// Mitsubishi GX Works2 project: Project-2   PLC: Q03UD

PROGRAM MAIN
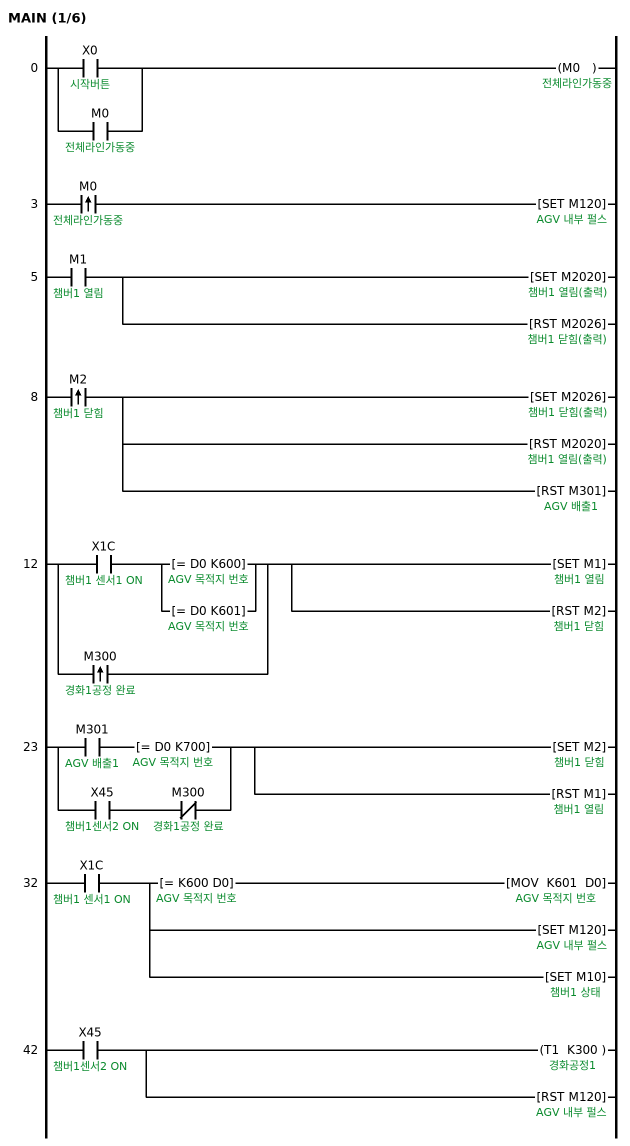
0     LD      X0  ; 시작버튼
      OR      M0  ; 전체라인가동중
      OUT     M0  ; 전체라인가동중
3     LDP     M0  ; 전체라인가동중
      SET     M120  ; AGV 내부 펄스
5     LD      M1  ; 챔버1 열림
      SET     M2020  ; 챔버1 열림(출력)
      RST     M2026  ; 챔버1 닫힘(출력)
8     LDP     M2  ; 챔버1 닫힘
      SET     M2026  ; 챔버1 닫힘(출력)
      RST     M2020  ; 챔버1 열림(출력)
      RST     M301  ; AGV 배출1
12    LD      X1C  ; 챔버1 센서1 ON
      LD=     D0 K600  ; AGV 목적지 번호
      OR=     D0 K601  ; AGV 목적지 번호
      ANB
      ORP     M300  ; 경화1공정 완료
      SET     M1  ; 챔버1 열림
      RST     M2  ; 챔버1 닫힘
23    LD      M301  ; AGV 배출1
      AND=    D0 K700  ; AGV 목적지 번호
      LD      X45  ; 챔버1센서2 ON
      ANI     M300  ; 경화1공정 완료
      ORB
      SET     M2  ; 챔버1 닫힘
      RST     M1  ; 챔버1 열림
32    LD      X1C  ; 챔버1 센서1 ON
      MPS
      AND=    K600 D0  ; AGV 목적지 번호
      MOV     K601 D0
      MPP
      SET     M120  ; AGV 내부 펄스
      SET     M10  ; 챔버1 상태
42    LD      X45  ; 챔버1센서2 ON
      OUT     T1 K300  ; 경화공정1
      RST     M120  ; AGV 내부 펄스
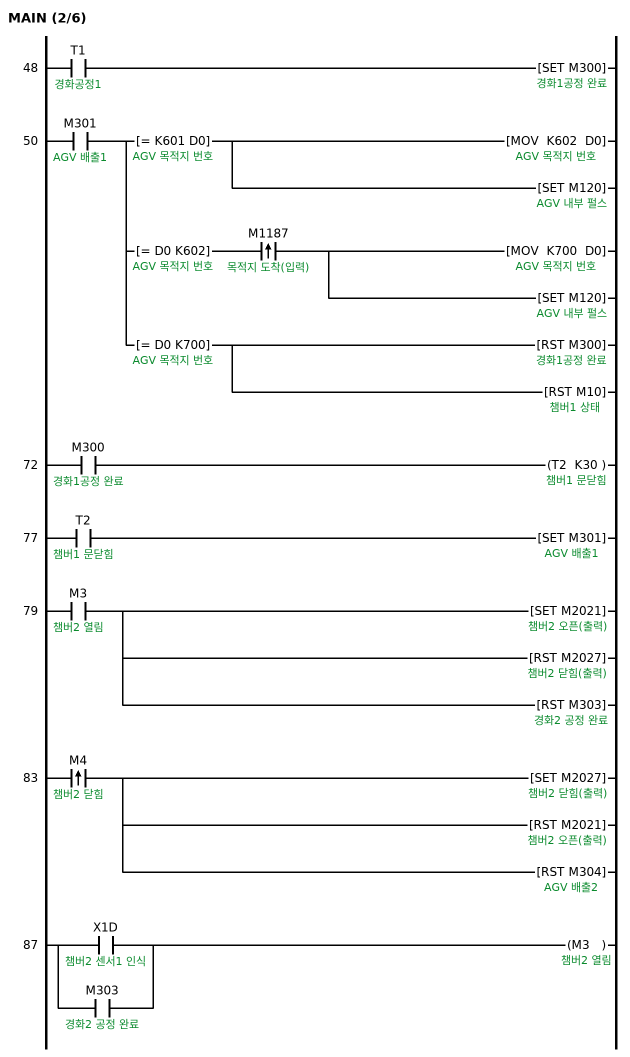
48    LD      T1  ; 경화공정1
      SET     M300  ; 경화1공정 완료
50    LD      M301  ; AGV 배출1
      MPS
      AND=    K601 D0  ; AGV 목적지 번호
      MOV     K602 D0
      SET     M120  ; AGV 내부 펄스
      MRD
      AND=    D0 K602  ; AGV 목적지 번호
      ANDP    M1187  ; 목적지 도착(입력)
      MOV     K700 D0
      SET     M120  ; AGV 내부 펄스
      MPP
      AND=    D0 K700  ; AGV 목적지 번호
      RST     M300  ; 경화1공정 완료
      RST     M10  ; 챔버1 상태
72    LD      M300  ; 경화1공정 완료
      OUT     T2 K30  ; 챔버1 문닫힘
77    LD      T2  ; 챔버1 문닫힘
      SET     M301  ; AGV 배출1
79    LD      M3  ; 챔버2 열림
      SET     M2021  ; 챔버2 오픈(출력)
      RST     M2027  ; 챔버2 닫힘(출력)
      RST     M303  ; 경화2 공정 완료
83    LDP     M4  ; 챔버2 닫힘
      SET     M2027  ; 챔버2 닫힘(출력)
      RST     M2021  ; 챔버2 오픈(출력)
      RST     M304  ; AGV 배출2
87    LD      X1D  ; 챔버2 센서1 인식
      OR      M303  ; 경화2 공정 완료
      OUT     M3  ; 챔버2 열림
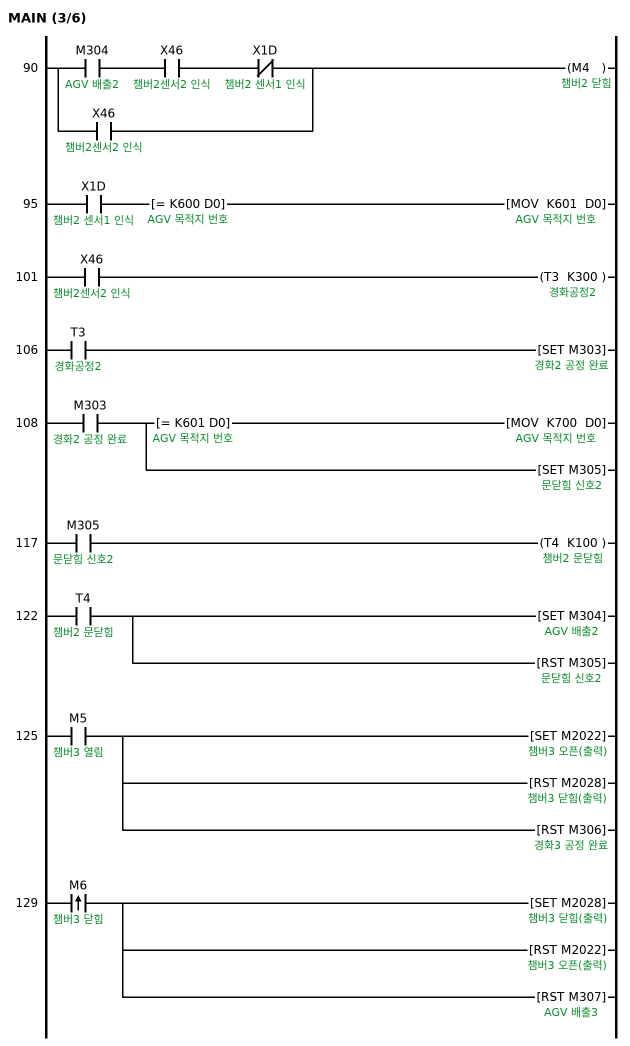
90    LD      M304  ; AGV 배출2
      AND     X46  ; 챔버2센서2 인식
      ANI     X1D  ; 챔버2 센서1 인식
      OR      X46  ; 챔버2센서2 인식
      OUT     M4  ; 챔버2 닫힘
95    LD      X1D  ; 챔버2 센서1 인식
      AND=    K600 D0  ; AGV 목적지 번호
      MOV     K601 D0
101   LD      X46  ; 챔버2센서2 인식
      OUT     T3 K300  ; 경화공정2
106   LD      T3  ; 경화공정2
      SET     M303  ; 경화2 공정 완료
108   LD      M303  ; 경화2 공정 완료
      MPS
      AND=    K601 D0  ; AGV 목적지 번호
      MOV     K700 D0
      MPP
      SET     M305  ; 문닫힘 신호2
117   LD      M305  ; 문닫힘 신호2
      OUT     T4 K100  ; 챔버2 문닫힘
122   LD      T4  ; 챔버2 문닫힘
      SET     M304  ; AGV 배출2
      RST     M305  ; 문닫힘 신호2
125   LD      M5  ; 챔버3 열림
      SET     M2022  ; 챔버3 오픈(출력)
      RST     M2028  ; 챔버3 닫힘(출력)
      RST     M306  ; 경화3 공정 완료
129   LDP     M6  ; 챔버3 닫힘
      SET     M2028  ; 챔버3 닫힘(출력)
      RST     M2022  ; 챔버3 오픈(출력)
      RST     M307  ; AGV 배출3
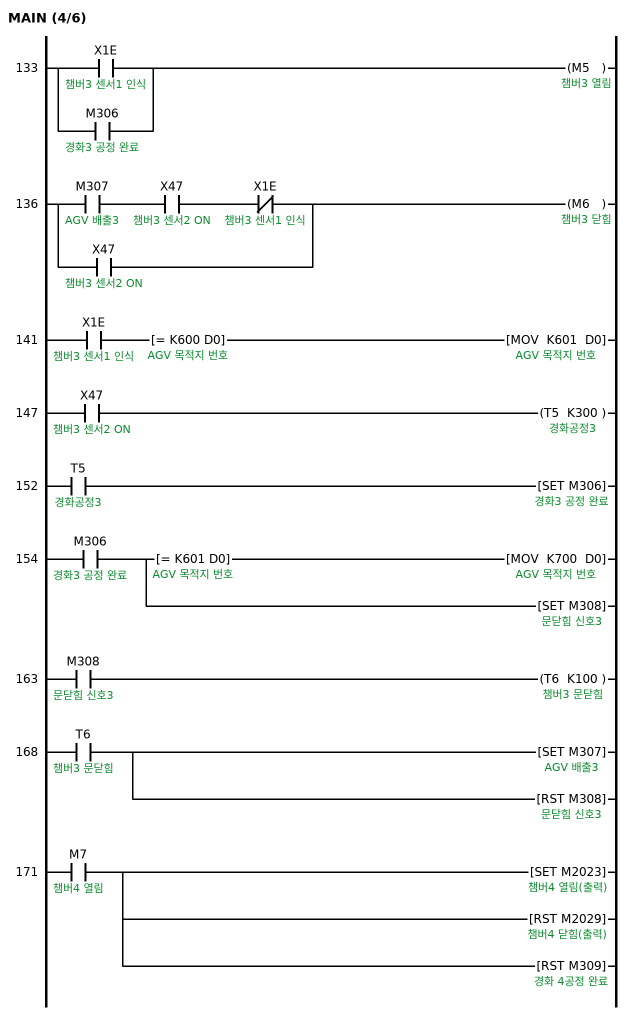
133   LD      X1E  ; 챔버3 센서1 인식
      OR      M306  ; 경화3 공정 완료
      OUT     M5  ; 챔버3 열림
136   LD      M307  ; AGV 배출3
      AND     X47  ; 챔버3 센서2 ON
      ANI     X1E  ; 챔버3 센서1 인식
      OR      X47  ; 챔버3 센서2 ON
      OUT     M6  ; 챔버3 닫힘
141   LD      X1E  ; 챔버3 센서1 인식
      AND=    K600 D0  ; AGV 목적지 번호
      MOV     K601 D0
147   LD      X47  ; 챔버3 센서2 ON
      OUT     T5 K300  ; 경화공정3
152   LD      T5  ; 경화공정3
      SET     M306  ; 경화3 공정 완료
154   LD      M306  ; 경화3 공정 완료
      MPS
      AND=    K601 D0  ; AGV 목적지 번호
      MOV     K700 D0
      MPP
      SET     M308  ; 문닫힘 신호3
163   LD      M308  ; 문닫힘 신호3
      OUT     T6 K100  ; 챔버3 문닫힘
168   LD      T6  ; 챔버3 문닫힘
      SET     M307  ; AGV 배출3
      RST     M308  ; 문닫힘 신호3
171   LD      M7  ; 챔버4 열림
      SET     M2023  ; 챔버4 열림(출력)
      RST     M2029  ; 챔버4 닫힘(출력)
      RST     M309  ; 경화 4공정 완료
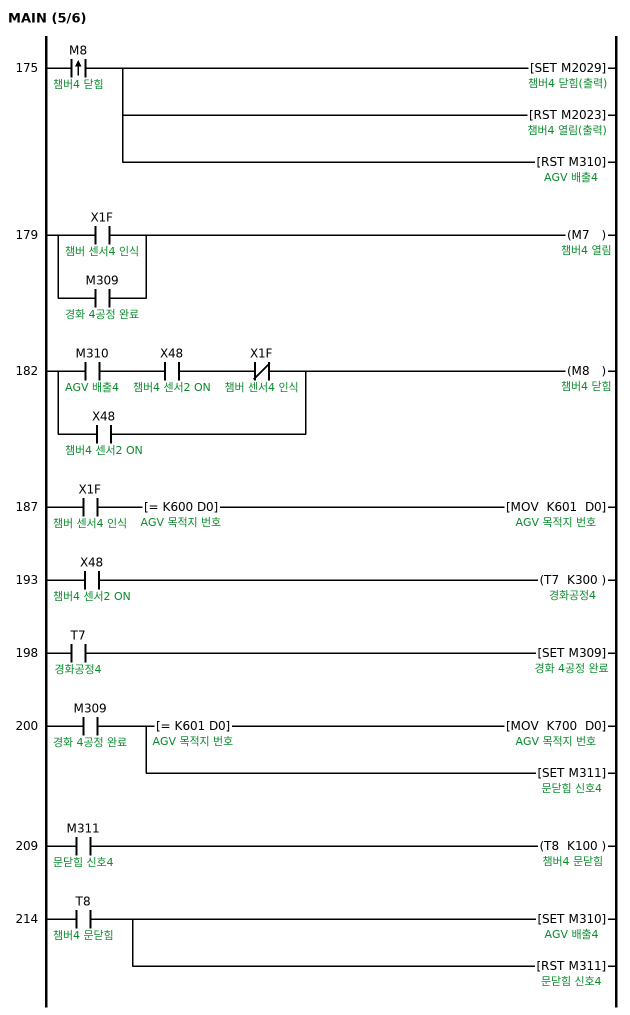
175   LDP     M8  ; 챔버4 닫힘
      SET     M2029  ; 챔버4 닫힘(출력)
      RST     M2023  ; 챔버4 열림(출력)
      RST     M310  ; AGV 배출4
179   LD      X1F  ; 챔버 센서4 인식
      OR      M309  ; 경화 4공정 완료
      OUT     M7  ; 챔버4 열림
182   LD      M310  ; AGV 배출4
      AND     X48  ; 챔버4 센서2 ON
      ANI     X1F  ; 챔버 센서4 인식
      OR      X48  ; 챔버4 센서2 ON
      OUT     M8  ; 챔버4 닫힘
187   LD      X1F  ; 챔버 센서4 인식
      AND=    K600 D0  ; AGV 목적지 번호
      MOV     K601 D0
193   LD      X48  ; 챔버4 센서2 ON
      OUT     T7 K300  ; 경화공정4
198   LD      T7  ; 경화공정4
      SET     M309  ; 경화 4공정 완료
200   LD      M309  ; 경화 4공정 완료
      MPS
      AND=    K601 D0  ; AGV 목적지 번호
      MOV     K700 D0
      MPP
      SET     M311  ; 문닫힘 신호4
209   LD      M311  ; 문닫힘 신호4
      OUT     T8 K100  ; 챔버4 문닫힘
214   LD      T8  ; 챔버4 문닫힘
      SET     M310  ; AGV 배출4
      RST     M311  ; 문닫힘 신호4
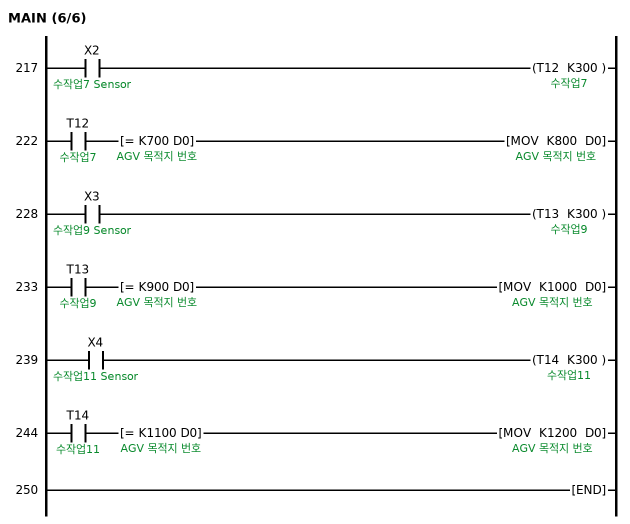
217   LD      X2  ; 수작업7 Sensor
      OUT     T12 K300  ; 수작업7
222   LD      T12  ; 수작업7
      AND=    K700 D0  ; AGV 목적지 번호
      MOV     K800 D0
228   LD      X3  ; 수작업9 Sensor
      OUT     T13 K300  ; 수작업9
233   LD      T13  ; 수작업9
      AND=    K900 D0  ; AGV 목적지 번호
      MOV     K1000 D0
239   LD      X4  ; 수작업11 Sensor
      OUT     T14 K300  ; 수작업11
244   LD      T14  ; 수작업11
      AND=    K1100 D0  ; AGV 목적지 번호
      MOV     K1200 D0
250   END
END_PROGRAM

PROGRAM AGV
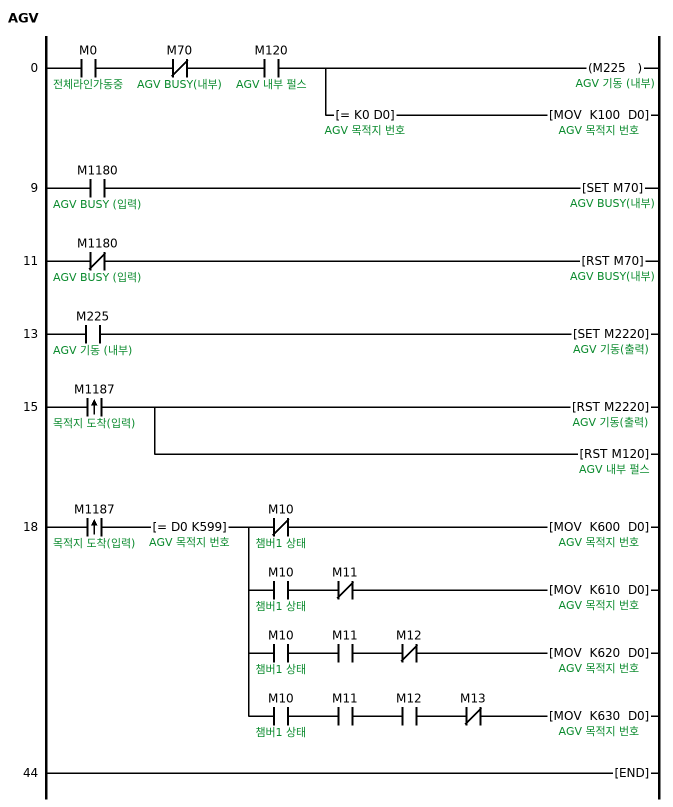
0     LD      M0  ; 전체라인가동중
      ANI     M70  ; AGV BUSY(내부)
      AND     M120  ; AGV 내부 펄스
      OUT     M225  ; AGV 기동 (내부)
      AND=    K0 D0  ; AGV 목적지 번호
      MOV     K100 D0
9     LD      M1180  ; AGV BUSY (입력)
      SET     M70  ; AGV BUSY(내부)
11    LDI     M1180  ; AGV BUSY (입력)
      RST     M70  ; AGV BUSY(내부)
13    LD      M225  ; AGV 기동 (내부)
      SET     M2220  ; AGV 기동(출력)
15    LDP     M1187  ; 목적지 도착(입력)
      RST     M2220  ; AGV 기동(출력)
      RST     M120  ; AGV 내부 펄스
18    LDP     M1187  ; 목적지 도착(입력)
      AND=    D0 K599  ; AGV 목적지 번호
      MPS
      ANI     M10  ; 챔버1 상태
      MOV     K600 D0
      MRD
      AND     M10  ; 챔버1 상태
      ANI     M11
      MOV     K610 D0
      MRD
      AND     M10  ; 챔버1 상태
      AND     M11
      ANI     M12
      MOV     K620 D0
      MPP
      AND     M10  ; 챔버1 상태
      AND     M11
      AND     M12
      ANI     M13
      MOV     K630 D0
44    END
END_PROGRAM

PROGRAM Rob1_1
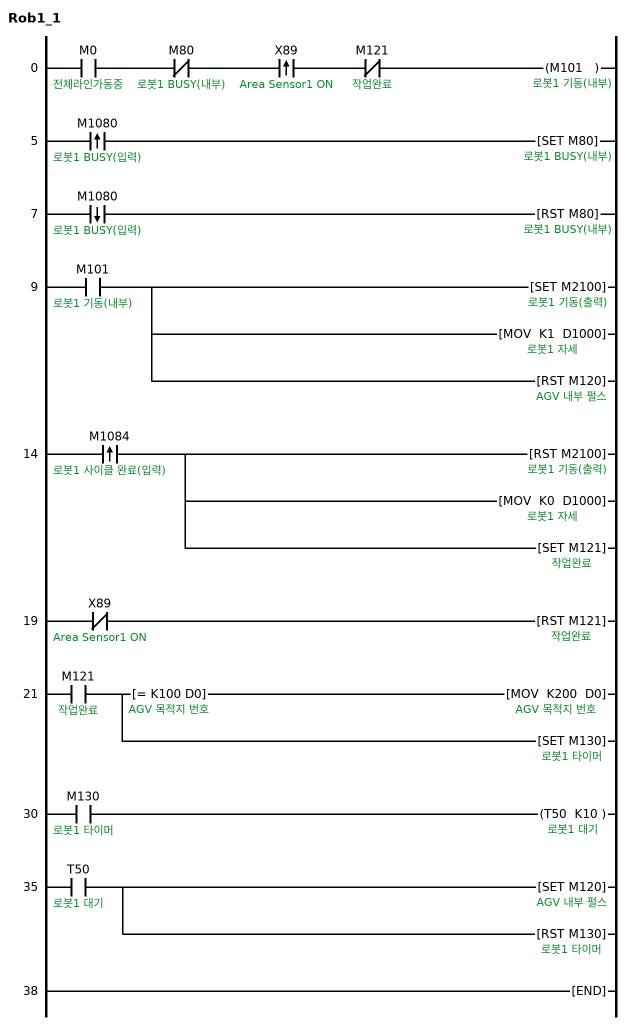
0     LD      M0  ; 전체라인가동중
      ANI     M80  ; 로봇1 BUSY(내부)
      ANDP    X89  ; Area Sensor1 ON
      ANI     M121  ; 작업완료
      OUT     M101  ; 로봇1 기동(내부)
5     LDP     M1080  ; 로봇1 BUSY(입력)
      SET     M80  ; 로봇1 BUSY(내부)
7     LDF     M1080  ; 로봇1 BUSY(입력)
      RST     M80  ; 로봇1 BUSY(내부)
9     LD      M101  ; 로봇1 기동(내부)
      SET     M2100  ; 로봇1 기동(출력)
      MOV     K1 D1000  ; 로봇1 자세
      RST     M120  ; AGV 내부 펄스
14    LDP     M1084  ; 로봇1 사이클 완료(입력)
      RST     M2100  ; 로봇1 기동(출력)
      MOV     K0 D1000
      SET     M121  ; 작업완료
19    LDI     X89  ; Area Sensor1 ON
      RST     M121  ; 작업완료
21    LD      M121  ; 작업완료
      MPS
      AND=    K100 D0  ; AGV 목적지 번호
      MOV     K200 D0
      MPP
      SET     M130  ; 로봇1 타이머
30    LD      M130  ; 로봇1 타이머
      OUT     T50 K10  ; 로봇1 대기
35    LD      T50  ; 로봇1 대기
      SET     M120  ; AGV 내부 펄스
      RST     M130  ; 로봇1 타이머
38    END
END_PROGRAM

PROGRAM Rob2_2
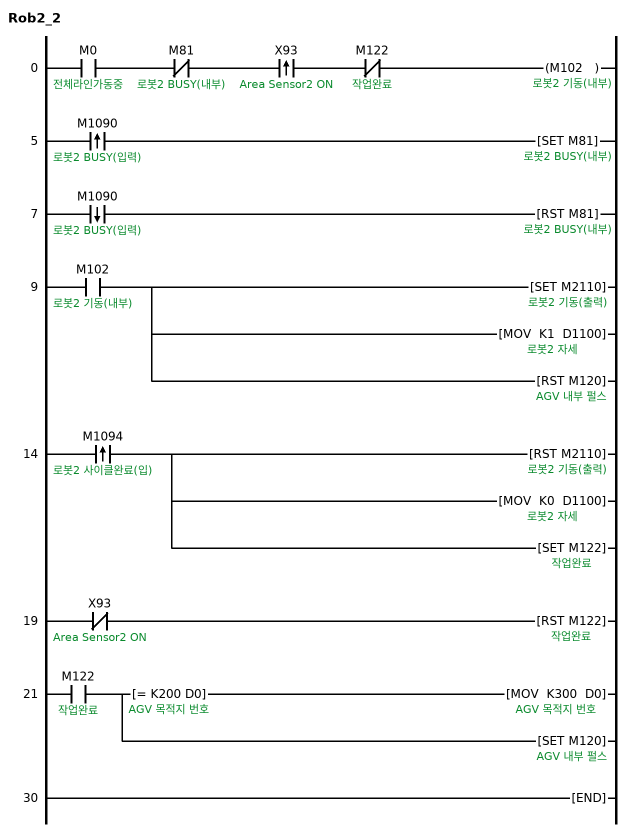
0     LD      M0  ; 전체라인가동중
      ANI     M81  ; 로봇2 BUSY(내부)
      ANDP    X93  ; Area Sensor2 ON
      ANI     M122  ; 작업완료
      OUT     M102  ; 로봇2 기동(내부)
5     LDP     M1090  ; 로봇2 BUSY(입력)
      SET     M81  ; 로봇2 BUSY(내부)
7     LDF     M1090  ; 로봇2 BUSY(입력)
      RST     M81  ; 로봇2 BUSY(내부)
9     LD      M102  ; 로봇2 기동(내부)
      SET     M2110  ; 로봇2 기동(출력)
      MOV     K1 D1100  ; 로봇2 자세
      RST     M120  ; AGV 내부 펄스
14    LDP     M1094  ; 로봇2 사이클완료(입)
      RST     M2110  ; 로봇2 기동(출력)
      MOV     K0 D1100
      SET     M122  ; 작업완료
19    LDI     X93  ; Area Sensor2 ON
      RST     M122  ; 작업완료
21    LD      M122  ; 작업완료
      MPS
      AND=    K200 D0  ; AGV 목적지 번호
      MOV     K300 D0
      MPP
      SET     M120  ; AGV 내부 펄스
30    END
END_PROGRAM

PROGRAM Rob3_3
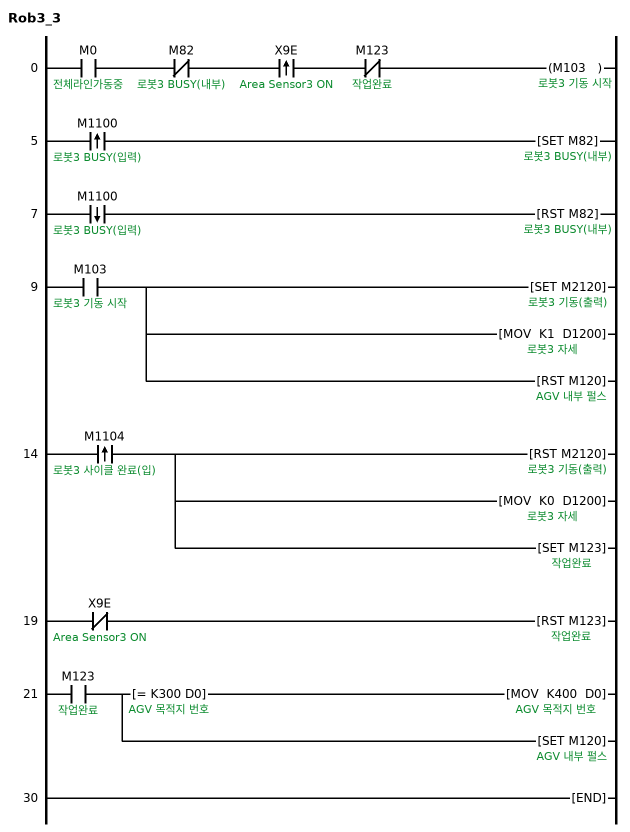
0     LD      M0  ; 전체라인가동중
      ANI     M82  ; 로봇3 BUSY(내부)
      ANDP    X9E  ; Area Sensor3 ON
      ANI     M123  ; 작업완료
      OUT     M103  ; 로봇3 기동 시작
5     LDP     M1100  ; 로봇3 BUSY(입력)
      SET     M82  ; 로봇3 BUSY(내부)
7     LDF     M1100  ; 로봇3 BUSY(입력)
      RST     M82  ; 로봇3 BUSY(내부)
9     LD      M103  ; 로봇3 기동 시작
      SET     M2120  ; 로봇3 기동(출력)
      MOV     K1 D1200  ; 로봇3 자세
      RST     M120  ; AGV 내부 펄스
14    LDP     M1104  ; 로봇3 사이클 완료(입)
      RST     M2120  ; 로봇3 기동(출력)
      MOV     K0 D1200
      SET     M123  ; 작업완료
19    LDI     X9E  ; Area Sensor3 ON
      RST     M123  ; 작업완료
21    LD      M123  ; 작업완료
      MPS
      AND=    K300 D0  ; AGV 목적지 번호
      MOV     K400 D0
      MPP
      SET     M120  ; AGV 내부 펄스
30    END
END_PROGRAM

PROGRAM Check_4
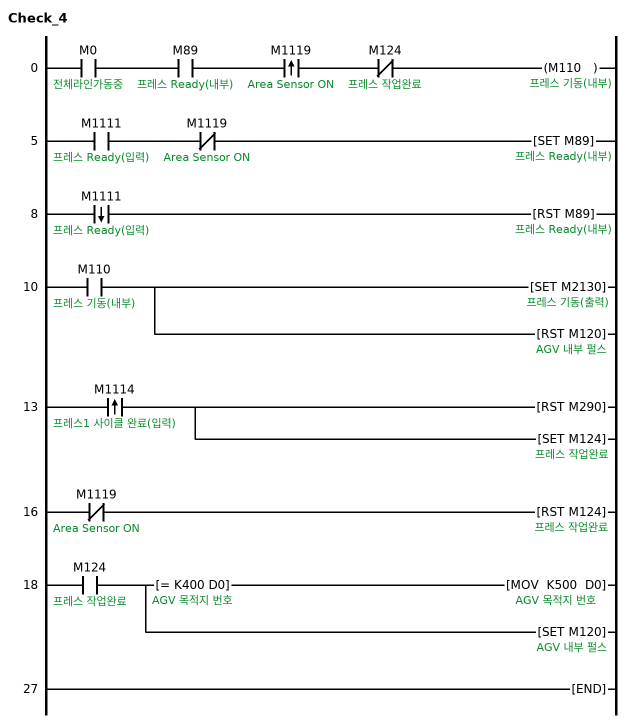
0     LD      M0  ; 전체라인가동중
      AND     M89  ; 프레스 Ready(내부)
      ANDP    M1119  ; Area Sensor ON
      ANI     M124  ; 프레스 작업완료
      OUT     M110  ; 프레스 기동(내부)
5     LD      M1111  ; 프레스 Ready(입력)
      ANI     M1119  ; Area Sensor ON
      SET     M89  ; 프레스 Ready(내부)
8     LDF     M1111  ; 프레스 Ready(입력)
      RST     M89  ; 프레스 Ready(내부)
10    LD      M110  ; 프레스 기동(내부)
      SET     M2130  ; 프레스 기동(출력)
      RST     M120  ; AGV 내부 펄스
13    LDP     M1114  ; 프레스1 사이클 완료(입력)
      RST     M290
      SET     M124  ; 프레스 작업완료
16    LDI     M1119  ; Area Sensor ON
      RST     M124  ; 프레스 작업완료
18    LD      M124  ; 프레스 작업완료
      MPS
      AND=    K400 D0  ; AGV 목적지 번호
      MOV     K500 D0
      MPP
      SET     M120  ; AGV 내부 펄스
27    END
END_PROGRAM

PROGRAM Rob5_5
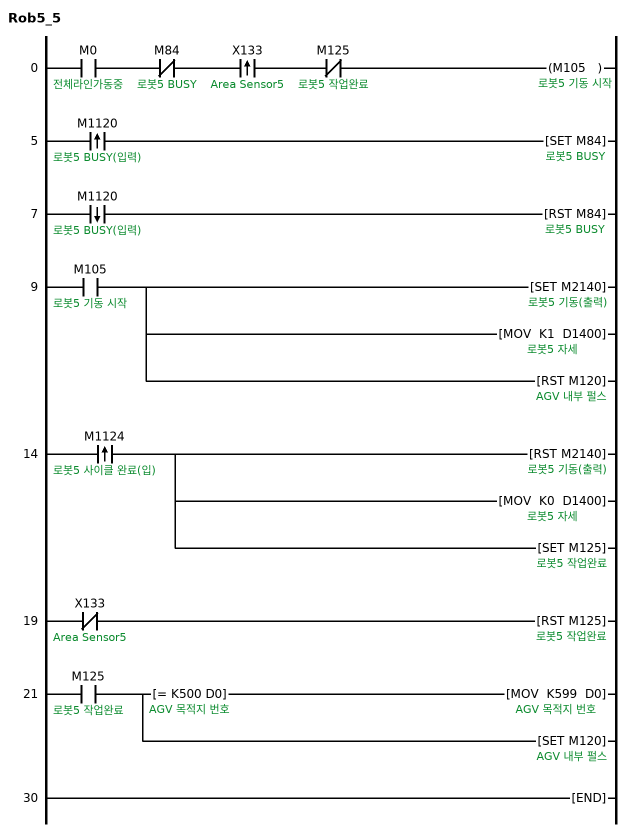
0     LD      M0  ; 전체라인가동중
      ANI     M84  ; 로봇5 BUSY
      ANDP    X133  ; Area Sensor5
      ANI     M125  ; 로봇5 작업완료
      OUT     M105  ; 로봇5 기동 시작
5     LDP     M1120  ; 로봇5 BUSY(입력)
      SET     M84  ; 로봇5 BUSY
7     LDF     M1120  ; 로봇5 BUSY(입력)
      RST     M84  ; 로봇5 BUSY
9     LD      M105  ; 로봇5 기동 시작
      SET     M2140  ; 로봇5 기동(출력)
      MOV     K1 D1400  ; 로봇5 자세
      RST     M120  ; AGV 내부 펄스
14    LDP     M1124  ; 로봇5 사이클 완료(입)
      RST     M2140  ; 로봇5 기동(출력)
      MOV     K0 D1400
      SET     M125  ; 로봇5 작업완료
19    LDI     X133  ; Area Sensor5
      RST     M125  ; 로봇5 작업완료
21    LD      M125  ; 로봇5 작업완료
      MPS
      AND=    K500 D0  ; AGV 목적지 번호
      MOV     K599 D0
      MPP
      SET     M120  ; AGV 내부 펄스
30    END
END_PROGRAM

PROGRAM Rob6_8
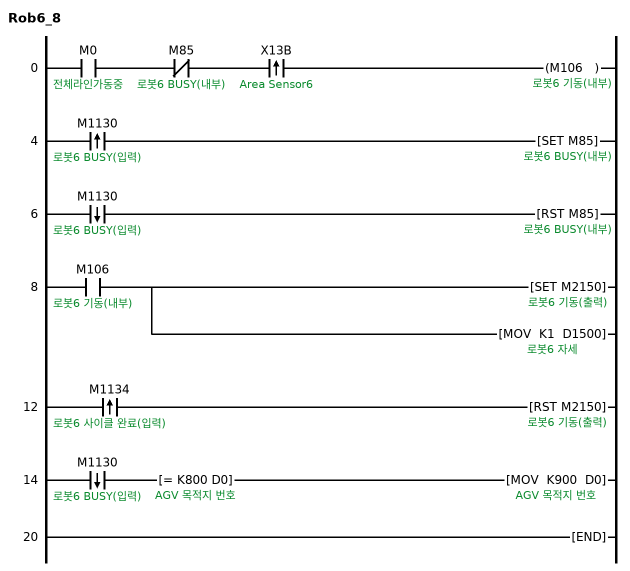
0     LD      M0  ; 전체라인가동중
      ANI     M85  ; 로봇6 BUSY(내부)
      ANDP    X13B  ; Area Sensor6
      OUT     M106  ; 로봇6 기동(내부)
4     LDP     M1130  ; 로봇6 BUSY(입력)
      SET     M85  ; 로봇6 BUSY(내부)
6     LDF     M1130  ; 로봇6 BUSY(입력)
      RST     M85  ; 로봇6 BUSY(내부)
8     LD      M106  ; 로봇6 기동(내부)
      SET     M2150  ; 로봇6 기동(출력)
      MOV     K1 D1500  ; 로봇6 자세
12    LDP     M1134  ; 로봇6 사이클 완료(입력)
      RST     M2150  ; 로봇6 기동(출력)
14    LDF     M1130  ; 로봇6 BUSY(입력)
      AND=    K800 D0  ; AGV 목적지 번호
      MOV     K900 D0
20    END
END_PROGRAM

PROGRAM Rob_12
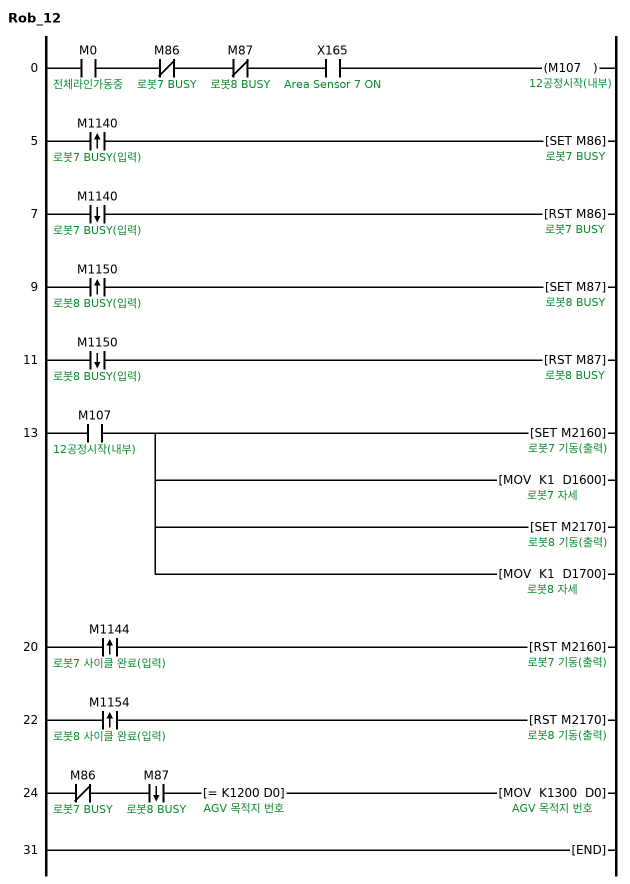
0     LD      M0  ; 전체라인가동중
      ANI     M86  ; 로봇7 BUSY
      ANI     M87  ; 로봇8 BUSY
      AND     X165  ; Area Sensor 7 ON
      OUT     M107  ; 12공정시작(내부)
5     LDP     M1140  ; 로봇7 BUSY(입력)
      SET     M86  ; 로봇7 BUSY
7     LDF     M1140  ; 로봇7 BUSY(입력)
      RST     M86  ; 로봇7 BUSY
9     LDP     M1150  ; 로봇8 BUSY(입력)
      SET     M87  ; 로봇8 BUSY
11    LDF     M1150  ; 로봇8 BUSY(입력)
      RST     M87  ; 로봇8 BUSY
13    LD      M107  ; 12공정시작(내부)
      SET     M2160  ; 로봇7 기동(출력)
      MOV     K1 D1600  ; 로봇7 자세
      SET     M2170  ; 로봇8 기동(출력)
      MOV     K1 D1700  ; 로봇8 자세
20    LDP     M1144  ; 로봇7 사이클 완료(입력)
      RST     M2160  ; 로봇7 기동(출력)
22    LDP     M1154  ; 로봇8 사이클 완료(입력)
      RST     M2170  ; 로봇8 기동(출력)
24    LDI     M86  ; 로봇7 BUSY
      ANDF    M87  ; 로봇8 BUSY
      AND=    K1200 D0  ; AGV 목적지 번호
      MOV     K1300 D0
31    END
END_PROGRAM

PROGRAM Rob9_13
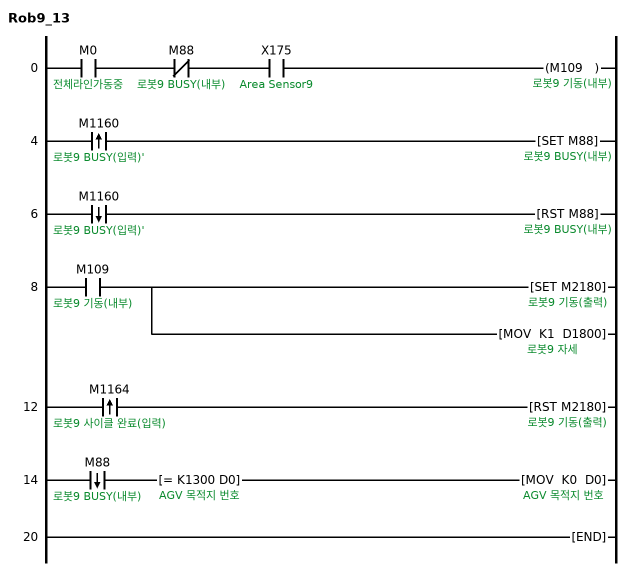
0     LD      M0  ; 전체라인가동중
      ANI     M88  ; 로봇9 BUSY(내부)
      AND     X175  ; Area Sensor9
      OUT     M109  ; 로봇9 기동(내부)
4     LDP     M1160  ; 로봇9 BUSY(입력)'
      SET     M88  ; 로봇9 BUSY(내부)
6     LDF     M1160  ; 로봇9 BUSY(입력)'
      RST     M88  ; 로봇9 BUSY(내부)
8     LD      M109  ; 로봇9 기동(내부)
      SET     M2180  ; 로봇9 기동(출력)
      MOV     K1 D1800  ; 로봇9 자세
12    LDP     M1164  ; 로봇9 사이클 완료(입력)
      RST     M2180  ; 로봇9 기동(출력)
14    LDF     M88  ; 로봇9 BUSY(내부)
      AND=    K1300 D0  ; AGV 목적지 번호
      MOV     K0 D0
20    END
END_PROGRAM

PROGRAM Press_10
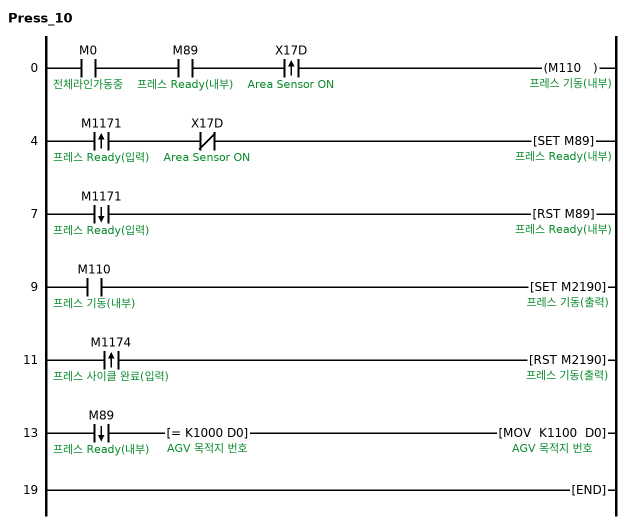
0     LD      M0  ; 전체라인가동중
      AND     M89  ; 프레스 Ready(내부)
      ANDP    X17D  ; Area Sensor ON
      OUT     M110  ; 프레스 기동(내부)
4     LDP     M1171  ; 프레스 Ready(입력)
      ANI     X17D  ; Area Sensor ON
      SET     M89  ; 프레스 Ready(내부)
7     LDF     M1171  ; 프레스 Ready(입력)
      RST     M89  ; 프레스 Ready(내부)
9     LD      M110  ; 프레스 기동(내부)
      SET     M2190  ; 프레스 기동(출력)
11    LDP     M1174  ; 프레스 사이클 완료(입력)
      RST     M2190  ; 프레스 기동(출력)
13    LDF     M89  ; 프레스 Ready(내부)
      AND=    K1000 D0  ; AGV 목적지 번호
      MOV     K1100 D0
19    END
END_PROGRAM

// device comments not shown above
X10  ; 로봇4 BUSY
X80  ; 로봇1 BUSY
X84  ; 로봇1 사이클 완료
X8A  ; 로봇2 BUSY
X8E  ; 로봇2 사이클 완료
X95  ; 로봇3 BUSY
X99  ; 로봇3 사이클 완료
X120  ; 로봇4 BUSY 신호
X124  ; 로봇4 사이클 완료
X129  ; Area Sensor4 ON
X12A  ; 로봇5 BUSY
X12E  ; 로봇5 사이클 완료
X132  ; 로봇6 BUSY
X136  ; 로봇6 사이클 완료
X13C  ; 로봇7 BUSY
X160  ; 로봇7 사이클 완료
X164  ; 로봇8 BUSY
X168  ; 로봇8 사이클 완료
X16C  ; 로봇9 BUSY
X170  ; 로봇9 사이클 완료
X17B  ; 프레스 Ready
X17E  ; 프레스 사이클 완료
X200  ; AGV BUSY
X201  ; AGV READY
X207  ; 도착완료
Y2  ; ㄹ
Y2D  ; 챔버1 열림
Y2E  ; 챔버2 열림
Y2F  ; 챔버3 열림
Y30  ; 챔버4 열림
Y71  ; 챔버1 닫기
Y72  ; 챔버2 닫기
Y73  ; 챔버3 닫기
Y74  ; 챔버 4 닫기
Y100  ; 로봇1 기동 시작
Y10A  ; 로봇2 기동 시작
Y115  ; 로봇3 기동 시작
Y140  ; 로봇4 기동 시작
Y14A  ; 로봇5 기동 시작
Y155  ; 로봇6 기동 시작
Y180  ; 로봇7 기동 시작
Y18A  ; 로봇8 기동 시작
Y193  ; 로봇9 기동 시작
Y19D  ; 프레스 기동 시작
Y225  ; AGV 기동 시작
M83  ; 로봇4 BUSY(내부)
M100  ; 로봇1 기동 시작
M104  ; 로봇4 기동 시작
M200  ; AGV BUSY
M302  ; 문닫힘신호1
M1110  ; 로봇4 BUSY(입력)
M1240  ; 로봇5 기동(출력)
D1  ; 1공정
D1300  ; 로봇4 자세
T0  ; 챔버 카운터
T9  ; 수작업7
T10  ; 수작업9
T11  ; 수작업11
T20  ; AGV 딜레이 신호
T101  ; 로봇1 대기
